// TIA Portal V16 export
// export: Created 2023-01-03T15:35:05.4721347Z, ExportSetting WithDefaults, DisplayName Totally Integrated Automation Portal, DisplayVersion V16, DisplayName TIA Portal Version Control Interface, DisplayVersion V16, DisplayName TIA Portal Openness, DisplayVersion V16, DisplayName STEP 7 Professional, DisplayVersion V16, DisplayName STEP 7 Safety, DisplayVersion V16, DisplayName WinCC Advanced, DisplayVersion V16
ORGANIZATION_BLOCK "Main"   // OB1, LAD, ProgramCycle
TITLE = "Main Program Sweep (Cycle)"
{ S7_Optimized_Access := 'TRUE' }
VERSION : 0.1
// stored: AutoNumber true, IsIECCheckEnabled false, SetENOAutomatically false
   VAR_INPUT
      Initial_Call : Bool;   // Initial call of this OB
      Remanence : Bool;   // =True, if remanent data are available
   END_VAR
   VAR_TEMP   // added for the SCL form of the ladder/FBD networks
      _w1 : Bool;
      _w2 : Bool;
   END_VAR
BEGIN

REGION Network 1: Main switch on
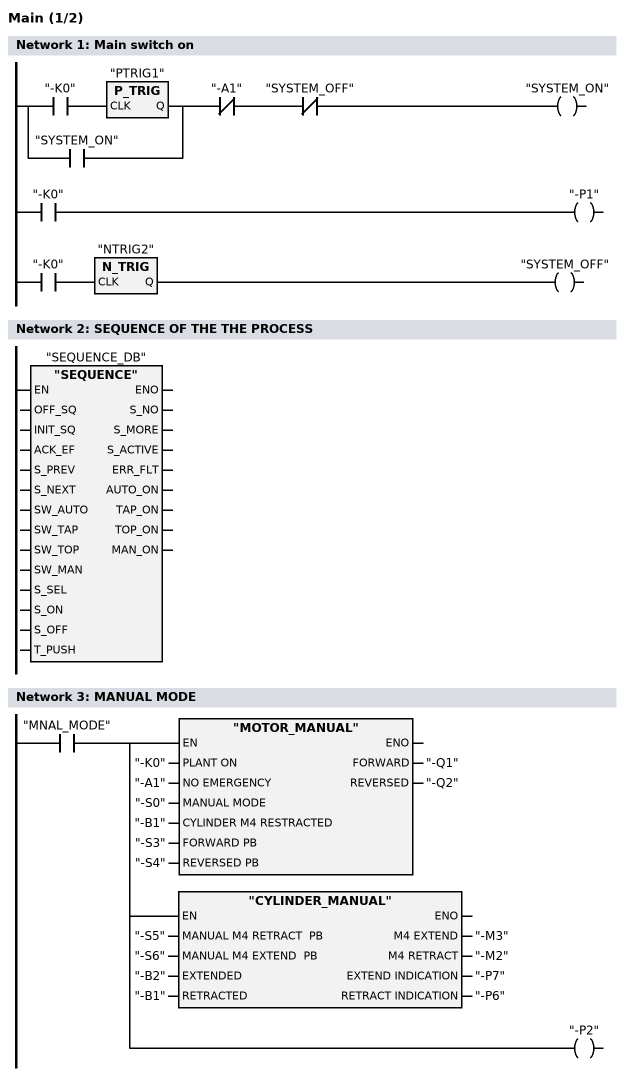
   RUNG wire#powerrail
      Contact( "-K0" )
      P_Trig( "PTRIG1" )
      wire#w1
      I_Contact( "-A1" )
      I_Contact( "SYSTEM_OFF" )
      Coil( "SYSTEM_ON" )
   END_RUNG
   RUNG wire#powerrail
      Contact( "SYSTEM_ON" )
   END_RUNG wire#w1
   RUNG wire#powerrail
      Contact( "-K0" )
      Coil( "-P1" )
   END_RUNG
   RUNG wire#powerrail
      Contact( "-K0" )
      N_Trig( "NTRIG2" )
      Coil( "SYSTEM_OFF" )
   END_RUNG
   // the same network as SCL:
   #_w1 := "-K0" AND NOT "PTRIG1";   // rising edge
   "PTRIG1" := "-K0";
   "SYSTEM_ON" := (#_w1 OR "SYSTEM_ON") AND NOT "-A1" AND NOT "SYSTEM_OFF";
   "-P1" := "-K0";
   #_w2 := NOT "-K0" AND "NTRIG2";   // falling edge
   "NTRIG2" := "-K0";
   "SYSTEM_OFF" := #_w2;
END_REGION

REGION Network 2: SEQUENCE OF THE THE PROCESS
   RUNG wire#powerrail
      "SEQUENCE_DB"(OFF_SQ :=, INIT_SQ :=, ACK_EF :=, S_PREV :=, S_NEXT :=, SW_AUTO :=, SW_TAP :=, SW_TOP :=, SW_MAN :=, S_SEL :=, S_ON :=, S_OFF :=, T_PUSH :=, S_NO =>, S_MORE =>, S_ACTIVE =>, ERR_FLT =>, AUTO_ON =>, TAP_ON =>, TOP_ON =>, MAN_ON =>)
   END_RUNG
   // the same network as SCL:
   "SEQUENCE_DB"();   // "SEQUENCE"
END_REGION

REGION Network 3: MANUAL MODE
   RUNG wire#powerrail
      Contact( "MNAL_MODE" )
      wire#w1
      "MOTOR_MANUAL"("PLANT ON" := "-K0", "NO EMERGENCY" := "-A1", "MANUAL MODE" := "-S0", "CYLINDER M4 RESTRACTED" := "-B1", "FORWARD PB" := "-S3", "REVERSED PB" := "-S4", FORWARD => "-Q1", REVERSED => "-Q2")
   END_RUNG
   RUNG wire#w1
      "CYLINDER_MANUAL"("MANUAL M4 RETRACT  PB" := "-S5", "MANUAL M4 EXTEND  PB" := "-S6", EXTENDED := "-B2", RETRACTED := "-B1", "M4 EXTEND" => "-M3", "M4 RETRACT" => "-M2", "EXTEND INDICATION" => "-P7", "RETRACT INDICATION" => "-P6")
   END_RUNG
   RUNG wire#w1
      Coil( "-P2" )
   END_RUNG
   // the same network as SCL:
   #_w1 := "MNAL_MODE";
   IF #_w1 THEN
       "MOTOR_MANUAL"("PLANT ON" := "-K0",
                      "NO EMERGENCY" := "-A1",
                      "MANUAL MODE" := "-S0",
                      "CYLINDER M4 RESTRACTED" := "-B1",
                      "FORWARD PB" := "-S3",
                      "REVERSED PB" := "-S4",
                      FORWARD => "-Q1",
                      REVERSED => "-Q2");
       "CYLINDER_MANUAL"("MANUAL M4 RETRACT  PB" := "-S5",
                         "MANUAL M4 EXTEND  PB" := "-S6",
                         EXTENDED := "-B2",
                         RETRACTED := "-B1",
                         "M4 EXTEND" => "-M3",
                         "M4 RETRACT" => "-M2",
                         "EXTEND INDICATION" => "-P7",
                         "RETRACT INDICATION" => "-P6");
   END_IF;
   "-P2" := #_w1;
END_REGION

REGION Network 4: AUTOMATIC MODE
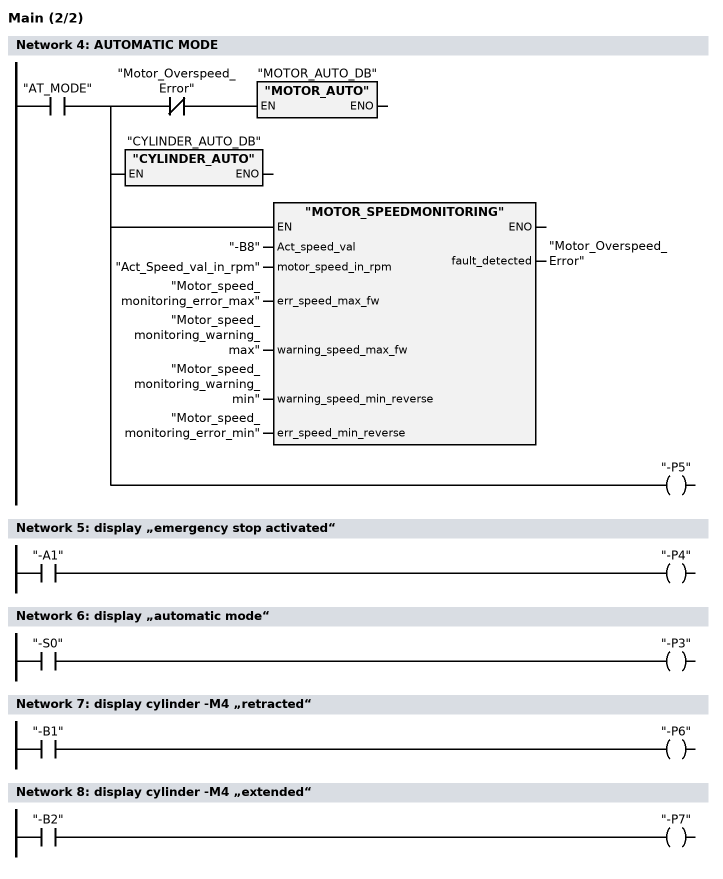
   RUNG wire#powerrail
      Contact( "AT_MODE" )
      wire#w1
      I_Contact( "Motor_Overspeed_Error" )
      "MOTOR_AUTO_DB"()
   END_RUNG
   RUNG wire#w1
      "CYLINDER_AUTO_DB"()
   END_RUNG
   RUNG wire#w1
      "MOTOR_SPEEDMONITORING"(Act_speed_val := "-B8", motor_speed_in_rpm := "Act_Speed_val_in_rpm", err_speed_max_fw := "Motor_speed_monitoring_error_max", warning_speed_max_fw := "Motor_speed_monitoring_warning_max", warning_speed_min_reverse := "Motor_speed_monitoring_warning_min", err_speed_min_reverse := "Motor_speed_monitoring_error_min", fault_detected => "Motor_Overspeed_Error")
   END_RUNG
   RUNG wire#w1
      Coil( "-P5" )
   END_RUNG
   // the same network as SCL:
   #_w1 := "AT_MODE";
   IF "AT_MODE" AND NOT "Motor_Overspeed_Error" THEN
       "MOTOR_AUTO_DB"();   // "MOTOR_AUTO"
   END_IF;
   IF #_w1 THEN
       "CYLINDER_AUTO_DB"();   // "CYLINDER_AUTO"
       "MOTOR_SPEEDMONITORING"(Act_speed_val := "-B8",
                               motor_speed_in_rpm := "Act_Speed_val_in_rpm",
                               err_speed_max_fw := "Motor_speed_monitoring_error_max",
                               warning_speed_max_fw := "Motor_speed_monitoring_warning_max",
                               warning_speed_min_reverse := "Motor_speed_monitoring_warning_min",
                               err_speed_min_reverse := "Motor_speed_monitoring_error_min",
                               fault_detected => "Motor_Overspeed_Error");
   END_IF;
   "-P5" := #_w1;
END_REGION

REGION Network 5: display „emergency stop activated“
   RUNG wire#powerrail
      Contact( "-A1" )
      Coil( "-P4" )
   END_RUNG
   // the same network as SCL:
   "-P4" := "-A1";
END_REGION

REGION Network 6: display „automatic mode“
   RUNG wire#powerrail
      Contact( "-S0" )
      Coil( "-P3" )
   END_RUNG
   // the same network as SCL:
   "-P3" := "-S0";
END_REGION

REGION Network 7: display cylinder -M4 „retracted“
   RUNG wire#powerrail
      Contact( "-B1" )
      Coil( "-P6" )
   END_RUNG
   // the same network as SCL:
   "-P6" := "-B1";
END_REGION

REGION Network 8: display cylinder -M4 „extended“
   RUNG wire#powerrail
      Contact( "-B2" )
      Coil( "-P7" )
   END_RUNG
   // the same network as SCL:
   "-P7" := "-B2";
END_REGION
END_ORGANIZATION_BLOCK
